// TIA Portal V20 export
TYPE "typeCmHmiInterface"
// stored: Access Published, Namespace Unit1.Em4
   STRUCT
      softcam : "Unit1.Em4.typeCmHmiInterfaceSoftCam";
   END_STRUCT;
END_TYPE
